PROGRAM VELOCIMETER
VAR
END_VAR

VelocimeterD := (RealVelocimeterD - VelocimeterSetPoint);

END_PROGRAM

(* stored: Version 1.1.0.1, ProductVersion 3.1.4024.12
   POU VELOCIMETER: Id {0b8ac552-5dca-4b11-a926-e1cfd53b31f2}, SpecialFunc None *)
